    {attribute 'pytmc' := '
    pv: ACTUAL_XWIDTH;
    io: io;
    '}
    rActApertureSizeX : REAL;

    {attribute 'pytmc' := '
    pv: ACTUAL_YWIDTH;
    io: io;
    '}
    rActApertureSizeY : REAL;
    {attribute 'pytmc' := '
    pv: ACTUAL_XCENTER;
    io: io;
    '}
    rActCenterX: REAL;
    {attribute 'pytmc' := '
    pv: ACTUAL_YCENTER;
    io: io;
    '}
    rActCenterY: REAL;

    {attribute 'pytmc' := '
    pv: XCEN_SETZERO;
    io: io;
    '}
    rSetCenterX: BOOL;
    {attribute 'pytmc' := '
    pv: YCEN_SETZERO;
    io: io;
    '}
    rSetCenterY: BOOL;


    {attribute 'pytmc' := '
    pv: OPEN;
    io: io;
    field: ZNAM False
    field: ONAM True
    '}
    bOpen: BOOL;

    {attribute 'pytmc' := '
    pv: CLOSE;
    io: io;
    field: ZNAM False
    field: ONAM True
    '}
    bClose: BOOL;

    {attribute 'pytmc' := '
    pv: BLOCK;
    io: io;
    field: ZNAM False
    field: ONAM True
    '}
    bBlock: BOOL;



        //Local variables
    bInit: BOOL :=true;
    rTrig_Block: R_TRIG;
    rTrig_Open: R_TRIG;
    rTrig_Close: R_TRIG;

    //old values
    rOldReqApertureSizeX : REAL;
    rOldReqApertureSizeY : REAL;
    rOldReqCenterX: REAL;
    rOldReqCenterY: REAL;

    bExecuteMotionX: BOOL;
    bExecuteMotionY: BOOL;


    fPosBlock: LREAL;
    fPosClose: LREAL;
    fPosOpen: LREAL;

    stSetPositionOptions:ST_SetPositionOptions;
    fbSetPosition_TOP: MC_SetPosition;
    fbSetPosition_Bottom: MC_SetPosition;
    fbSetPosition_North: MC_SetPosition;
    fbSetPosition_South: MC_SetPosition;

    // For logging
    fbLogger : FB_LogMessage := (eSubsystem:=E_SubSystem.MOTION);
    tErrorPresent : R_TRIG;
    tAction : R_TRIG;
    tOverrideActivated : R_TRIG;

    FFO    :    FB_FastFault :=(
        i_DevName := 'Slits',
        i_Desc := 'Fault occurs when gaps and/or centers are not within safe margins, or PMPS mode is switched OFF',
        i_TypeCode := 16#FAA);

    AptArrayStatus AT %Q* : ST_PMPS_Aperture_IO;
    AptArrayReq AT %I* : ST_PMPS_Aperture_IO;

    bTest: BOOL;

END_VAR

ACTION ACT_BLOCK:
rTrig_Block (CLK:= bBlock);
rTrig_Open (CLK:= bOpen);
rTrig_Close (CLK:= bClose);

if (rTrig_Block.Q) THEN
    //BLOCK

    bBlock := false;
END_IF

if (rTrig_Open.Q) THEN


    bOpen := false;
END_IF

if (rTrig_Close.Q) THEN


    bClose := false;
END_IF
END_ACTION

ACTION ACT_CalculatePositions:
//check if requested center or gap has changed
//check that the requested values are within acceptable motion range
IF (rOldReqApertureSizeX <> rReqApertureSizeX) THEN
    IF (rReqApertureSizeX <= AptArrayReq.Width)  THEN
        rOldReqApertureSizeX := rReqApertureSizeX;
        bExecuteMotionX := TRUE;
        fbLogger(sMsg:='Requested new X gap.', eSevr:=TcEventSeverity.Verbose);
    ELSE
        fbLogger(sMsg:='Requested new X gap is larger than PMPS request.', eSevr:=TcEventSeverity.Verbose);
    END_IF
  //  ELSE
    //    rReqApertureSizeX := rActApertureSizeX;
END_IF

IF (rOldReqCenterX <> rReqCenterX) THEN
    rOldReqCenterX := rReqCenterX;
    bExecuteMotionX := TRUE;
    fbLogger(sMsg:='Requested new X center', eSevr:=TcEventSeverity.Verbose);
   // ELSE
      //  rReqCenterX := rActCenterX;
END_IF

IF (rOldReqApertureSizeY <> rReqApertureSizeY) THEN
    IF rReqApertureSizeY <= AptArrayReq.Height THEN
        rOldReqApertureSizeY := rReqApertureSizeY;
        bExecuteMotionY := TRUE;
        fbLogger(sMsg:='Requested new Y gap.', eSevr:=TcEventSeverity.Verbose);
    ELSE
        fbLogger(sMsg:='Requested new Y gap is larger than PMPS request.', eSevr:=TcEventSeverity.Verbose);
    END_IF
   // ELSE
       // rReqApertureSizeY := rActApertureSizeY;
END_IF

IF (rOldReqCenterY <> rReqCenterY) THEN
    rOldReqCenterY := rReqCenterY;
    bExecuteMotionY := TRUE;
    fbLogger(sMsg:='Requested new Y center.', eSevr:=TcEventSeverity.Verbose);
   // ELSE
      //  rReqCenterY := rActCenterY;
END_IF


//Calculate requested target positions from requested gap and center
fPosTopBlade := (rReqApertureSizeY/2) + (rReqCenterY + rEncoderOffsetTop) ;
fPosBottomBlade := (-1*rReqApertureSizeY/2) + (rReqCenterY+rEncoderOffsetBottom);

fPosNorthBlade := (rReqApertureSizeX/2) + (rReqCenterX + rEncoderOffsetNorth);
fPosSouthBlade := (-1*rReqApertureSizeX/2) + (rReqCenterX + rEncoderOffsetSouth);


//Calculate actual gap and center from actual stages positions
rActApertureSizeX := LREAL_TO_REAL((stNorthBlade.stAxisStatus.fActPosition - rEncoderOffsetNorth) - (stSouthBlade.stAxisStatus.fActPosition- rEncoderOffsetSouth));

rActApertureSizeY := LREAL_TO_REAL((stTopBlade.stAxisStatus.fActPosition - rEncoderOffsetTop) - (stBottomBlade.stAxisStatus.fActPosition - rEncoderOffsetBottom));

rActCenterX := LREAL_TO_REAL((((stNorthBlade.stAxisStatus.fActPosition - rEncoderOffsetNorth)  + (stSouthBlade.stAxisStatus.fActPosition - rEncoderOffsetSouth ))/2));

rActCenterY := LREAL_TO_REAL((((stTopBlade.stAxisStatus.fActPosition - rEncoderOffsetTop) + (stBottomBlade.stAxisStatus.fActPosition - rEncoderOffsetBottom))/2));



//Update PMPS Arbiter with the Actual Size and Center of the Aperture
END_ACTION

ACTION ACT_Home:

END_ACTION

ACTION ACT_Init:

//  init the motion stages parameters
IF ( bInit) THEN
    stTopBlade.bHardwareEnable := TRUE;
    stBottomBlade.bHardwareEnable := TRUE;
    stNorthBlade.bHardwareEnable := TRUE;
    stSouthBlade.bHardwareEnable := TRUE;
    stTopBlade.bPowerSelf :=TRUE;
    stBottomBlade.bPowerSelf :=TRUE;
    stNorthBlade.bPowerSelf :=TRUE;
    stSouthBlade.bPowerSelf :=TRUE;
    stTopBlade.nBrakeMode := ENUM_StageBrakeMode.NO_BRAKE;
    stBottomBlade.nBrakeMode := ENUM_StageBrakeMode.NO_BRAKE;
    stNorthBlade.nBrakeMode := ENUM_StageBrakeMode.NO_BRAKE;
    stSouthBlade.nBrakeMode := ENUM_StageBrakeMode.NO_BRAKE;
    FFO.i_DevName := i_DevName;
END_IF
END_ACTION

ACTION ACT_Motion:
// Instantiate Function block for all the blades
fbTopBlade(stMotionStage:=stTopBlade);
fbBottomBlade(stMotionStage:=stBottomBlade);
fbNorthBlade(stMotionStage:=stNorthBlade);
fbSouthBlade(stMotionStage:=stSouthBlade);

// PTP Motion for each blade
stTop.sName := 'Top';
stTop.fPosition := fPosTopBlade;
stTop.fDelta := fSmallDelta;
stTop.fVelocity := fMaxVelocity;
stTop.fAccel := fHighAccel;
stTop.fDecel := fHighAccel;

stBOTTOM.sName := 'Bottom';
stBOTTOM.fPosition := fPosBottomBlade;
stBOTTOM.fDelta := fSmallDelta;
stBOTTOM.fVelocity := fMaxVelocity;
stBOTTOM.fAccel := fHighAccel;
stBOTTOM.fDecel := fHighAccel;

stNorth.sName := 'North';
stNorth.fPosition := fPosNorthBlade;
stNorth.fDelta := fSmallDelta;
stNorth.fVelocity := fMaxVelocity;
stNorth.fAccel := fHighAccel;
stNorth.fDecel := fHighAccel;

stSouth.sName := 'South';
stSouth.fPosition := fPosSouthBlade;
stSouth.fDelta := fSmallDelta;
stSouth.fVelocity := fMaxVelocity;
stSouth.fAccel := fHighAccel;
stSouth.fDecel := fHighAccel;

IF (bExecuteMotionY) THEN
    fbTop.bExecute := fbBottom.bExecute := bExecuteMotionY;
    bExecuteMotionY:= FALSE;
END_IF

IF (bExecuteMotionX) THEN
    fbNorth.bExecute := fbSouth.bExecute := bExecuteMotionX;
    bExecuteMotionX:= FALSE;
END_IF


fbTop(
    stPositionState:=stTop,
    bMoveOk:=bMoveOk,
    stMotionStage:=stTopBlade);

fbBottom(
    stPositionState:=stBOTTOM,
    bMoveOk:=bMoveOk,
    stMotionStage:=stBottomBlade);

fbNorth(
    stPositionState:=stNorth,
    bMoveOk:=bMoveOk,
    stMotionStage:=stNorthBlade);

fbSouth(
    stPositionState:=stSouth,
    bMoveOk:=bMoveOk,
    stMotionStage:=stSouthBlade);
END_ACTION

ACTION ACT_Zero:
//ZERO BIAS

// Set Y center to zero

// Set X center to zero
(*
if (rSetCenterY)THEN
        rSetCenterY := false;
        // Set Current Position
        fbSetPosition_TOP.Position :=  stTopBlade.stAxisStatus.fActPosition - rActCenterY ;
        fbSetPosition_TOP.Execute := TRUE;
        fbSetPosition_Bottom.Position := stBottomBlade.stAxisStatus.fActPosition - rActCenterY;
        fbSetPosition_Bottom.Execute := TRUE;
END_IF

if (rSetCenterX)THEN
        rSetCenterX := false;
        // Set Current Position
        fbSetPosition_North.Position := stNorthBlade.stAxisStatus.fActPosition - rActCenterX ;
        fbSetPosition_North.Execute := TRUE;
        fbSetPosition_South.Position := stSouthBlade.stAxisStatus.fActPosition - rActCenterX ; ;
        fbSetPosition_South.Execute := TRUE;
END_IF


//Reset
if (fbSetPosition_TOP.Done ) THEN
    fbSetPosition_TOP.Execute := FALSE;
END_IF
if (fbSetPosition_Bottom.Done ) THEN
    fbSetPosition_Bottom.Execute := FALSE;
END_IF
if (fbSetPosition_North.Done ) THEN
    fbSetPosition_North.Execute := FALSE;
END_IF
if (fbSetPosition_South.Done ) THEN
    fbSetPosition_South.Execute := FALSE;
END_IF

// Set Encoder Position
//Clear position lag error
stSetPositionOptions.ClearPositionLag := TRUE;
fbSetPosition_TOP(
    Axis:=  stTopBlade.Axis ,
    Execute:= ,
    Position:= 0 ,
    Mode:= FALSE,
    Options:= stSetPositionOptions,
    Done=> ,
    Busy=> ,
    Error=> ,
    ErrorID=> );
fbSetPosition_Bottom(
    Axis:= stBottomBlade.Axis ,
    Execute:= ,
    Position:= 0 ,
    Mode:= FALSE,
    Options:= stSetPositionOptions,
    Done=> ,
    Busy=> ,
    Error=> ,
    ErrorID=> );
fbSetPosition_North(
    Axis:= stNorthBlade.Axis ,
    Execute:= ,
    Position:= 0 ,
    Mode:= FALSE,
    Options:= stSetPositionOptions,
    Done=> ,
    Busy=> ,
    Error=> ,
    ErrorID=> );
fbSetPosition_South(
    Axis:= stSouthBlade.Axis ,
    Execute:= ,
    Position:= 0 ,
    Mode:= FALSE,
    Options:= stSetPositionOptions,
    Done=> ,
    Busy=> ,
    Error=> ,
    ErrorID=> );

    *)
END_ACTION

END_FUNCTION_BLOCK

// ---- POUs/PRG_SL2K0_POWER.TcPOU
PROGRAM PRG_SL2K0_POWER
VAR
    {attribute 'pytmc' := '
        pv: SL2K0:POWER
        io: io
    '}
    {attribute 'TcLinkTo' := '.RTD_South_1.iRaw := TIIB[SL2K0-EL3202-E8]^RTD Inputs Channel 1^Value;
                              .RTD_South_1.bError := TIIB[SL2K0-EL3202-E8]^RTD Inputs Channel 1^Status^Error;
                              .RTD_South_1.bUnderrange := TIIB[SL2K0-EL3202-E8]^RTD Inputs Channel 1^Status^Underrange;
                              .RTD_South_1.bOverrange := TIIB[SL2K0-EL3202-E8]^RTD Inputs Channel 1^Status^Overrange;
                              .RTD_South_2.iRaw := TIIB[SL2K0-EL3202-E8]^RTD Inputs Channel 2^Value;
                              .RTD_South_2.bError := TIIB[SL2K0-EL3202-E8]^RTD Inputs Channel 2^Status^Error;
                              .RTD_South_2.bUnderrange := TIIB[SL2K0-EL3202-E8]^RTD Inputs Channel 2^Status^Underrange;
                              .RTD_South_2.bOverrange := TIIB[SL2K0-EL3202-E8]^RTD Inputs Channel 2^Status^Overrange;
                              .RTD_TOP_1.iRaw := TIIB[SL2K0-EL3202-E9]^RTD Inputs Channel 1^Value;
                              .RTD_TOP_1.bError := TIIB[SL2K0-EL3202-E9]^RTD Inputs Channel 1^Status^Error;
                              .RTD_TOP_1.bUnderrange := TIIB[SL2K0-EL3202-E9]^RTD Inputs Channel 1^Status^Underrange;
                              .RTD_TOP_1.bOverrange := TIIB[SL2K0-EL3202-E9]^RTD Inputs Channel 1^Status^Overrange;
                              .RTD_TOP_2.iRaw := TIIB[SL2K0-EL3202-E9]^RTD Inputs Channel 2^Value;
                              .RTD_TOP_2.bError := TIIB[SL2K0-EL3202-E9]^RTD Inputs Channel 2^Status^Error;
                              .RTD_TOP_2.bUnderrange := TIIB[SL2K0-EL3202-E9]^RTD Inputs Channel 2^Status^Underrange;
                              .RTD_TOP_2.bOverrange := TIIB[SL2K0-EL3202-E9]^RTD Inputs Channel 2^Status^Overrange;
                              .RTD_North_1.iRaw := TIIB[SL2K0-EL3202-E10]^RTD Inputs Channel 1^Value;
                              .RTD_North_1.bError := TIIB[SL2K0-EL3202-E10]^RTD Inputs Channel 1^Status^Error;
                              .RTD_North_1.bUnderrange := TIIB[SL2K0-EL3202-E10]^RTD Inputs Channel 1^Status^Underrange;
                              .RTD_North_1.bOverrange := TIIB[SL2K0-EL3202-E10]^RTD Inputs Channel 1^Status^Overrange;
                              .RTD_North_2.iRaw := TIIB[SL2K0-EL3202-E10]^RTD Inputs Channel 2^Value;
                              .RTD_North_2.bError := TIIB[SL2K0-EL3202-E10]^RTD Inputs Channel 2^Status^Error;
                              .RTD_North_2.bUnderrange := TIIB[SL2K0-EL3202-E10]^RTD Inputs Channel 2^Status^Underrange;
                              .RTD_North_2.bOverrange := TIIB[SL2K0-EL3202-E10]^RTD Inputs Channel 2^Status^Overrange;
                              .RTD_Bottom_1.iRaw := TIIB[SL2K0-EL3202-E10]^RTD Inputs Channel 1^Value;
                              .RTD_Bottom_1.bError := TIIB[SL2K0-EL3202-E10]^RTD Inputs Channel 1^Status^Error;
                              .RTD_Bottom_1.bUnderrange := TIIB[SL2K0-EL3202-E11]^RTD Inputs Channel 1^Status^Underrange;
                              .RTD_Bottom_1.bOverrange := TIIB[SL2K0-EL3202-E11]^RTD Inputs Channel 1^Status^Overrange;
                              .RTD_Bottom_2.iRaw := TIIB[SL2K0-EL3202-E11]^RTD Inputs Channel 2^Value;
                              .RTD_Bottom_2.bError := TIIB[SL2K0-EL3202-E11]^RTD Inputs Channel 2^Status^Error;
                              .RTD_Bottom_2.bUnderrange := TIIB[SL2K0-EL3202-E11]^RTD Inputs Channel 2^Status^Underrange;
                              .RTD_Bottom_2.bOverrange := TIIB[SL2K0-EL3202-E11]^RTD Inputs Channel 2^Status^Overrange;
                              .AptArrayStatus := TIIB[PMPS_PRE]^IO Outputs^AptArrayStatus^AptArrayStatus[2];
                              .AptArrayReq := TIIB[PMPS_PRE]^IO Inputs^AptArrayReq^AptArrayReq[2];
                              .fbFlowSwitch.bFlowOk := TIIB[SL2K0-EL1004-E12]^Channel 1^Input'}
    fbSL2K0: FB_SLITS_POWER;
//GET PMP Move Ok bit
// Default True until it is properly linked to PMPS bit
    bMoveOk:BOOL :=TRUE;
    {attribute 'pytmc' := '
    pv: SL2K0:POWER:GO;
    io: io;
    field: ZNAM False;
    field: ONAM True;
    '}
    bExecuteMotion:BOOL ;
    //for testing purposes only. comment-out/delete once done.
    mcPower : ARRAY [1..4] OF MC_POWER;
        (*Offsets*)
    (* Absolute encoder value at the HLS + Absolure eoncoder value at the centered beam *)
    rEncoderOffsetTop: REAL := 14.65; //15.1;
    rEncoderOffsetBottom: REAL := -12.55; //-12.2;
    rEncoderOffsetNorth: REAL :=  16.3; //15.4;
    rEncoderOffsetSouth: REAL := -12.94; //-13.4;
END_VAR


fbSL2K0.bMoveOk := bMoveOk;

fbSL2K0.rEncoderOffsetTop := rEncoderOffsetTop;
fbSL2K0.rEncoderOffsetBottom := rEncoderOffsetBottom;
fbSL2K0.rEncoderOffsetNorth := rEncoderOffsetNorth;
fbSL2K0.rEncoderOffsetSouth := rEncoderOffsetSouth;

fbSL2K0(stTopBlade:=  Main.M23,
        stBottomBlade:= Main.M25,
        stNorthBlade:=  Main.M24,
        stSouthBlade:=  Main.M22,
        bExecuteMotion:=bExecuteMotion,
        io_fbFFHWO := GVL.fbFastFaultOutput1,
        fbArbiter := GVL.fbArbiter);

fbSL2K0.M_UpdatePMPS(2);


//for testing purposes only. comment-out/delete once done.
(*mcPower[1](axis:=Main.M22.Axis, Enable:=TRUE, enable_positive:=Main.M22.bLimitForwardEnable, enable_negative:=Main.M22.bLimitBackwardEnable);
mcPower[2](axis:=Main.M23.Axis, Enable:=TRUE, enable_positive:=Main.M23.bLimitForwardEnable, enable_negative:=Main.M23.bLimitBackwardEnable);
mcPower[3](axis:=Main.M24.Axis, Enable:=TRUE, enable_positive:=Main.M24.bLimitForwardEnable, enable_negative:=Main.M24.bLimitBackwardEnable);
mcPower[4](axis:=Main.M25.Axis, Enable:=TRUE, enable_positive:=Main.M25.bLimitForwardEnable, enable_negative:=Main.M25.bLimitBackwardEnable);*)

END_PROGRAM

// ---- POUs/PRG_AT1K4_SOLID.TcPOU
PROGRAM PRG_AT1K4_SOLID
VAR
    (* TODO: use FALSE for simulation and production *)
    (* TODO: use TRUE when relying on visualization + actual hardware *)
    bDebug : BOOL := FALSE;

    nEnableMode : ENUM_StageEnableMode;

    {attribute 'pytmc' := 'pv: AT1K4:L2SI:MMS:01'}
    {attribute 'TcLinkTo' := '

        .fbRTD_1.iRaw := TIIB[AT1K4-EL3202-04]^RTD Inputs Channel 1^Value;
        .fbRTD_1.bError := TIIB[AT1K4-EL3202-04]^RTD Inputs Channel 1^Status^Error;
        .fbRTD_1.bUnderrange := TIIB[AT1K4-EL3202-04]^RTD Inputs Channel 1^Status^Underrange;
        .fbRTD_1.bOverrange := TIIB[AT1K4-EL3202-04]^RTD Inputs Channel 1^Status^Overrange;

        .fbRTD_2.iRaw := TIIB[AT1K4-EL3202-04]^RTD Inputs Channel 2^Value;
        .fbRTD_2.bError := TIIB[AT1K4-EL3202-04]^RTD Inputs Channel 2^Status^Error;
        .fbRTD_2.bUnderrange := TIIB[AT1K4-EL3202-04]^RTD Inputs Channel 2^Status^Underrange;
        .fbRTD_2.bOverrange := TIIB[AT1K4-EL3202-04]^RTD Inputs Channel 2^Status^Overrange

    '}
    fbStage1: FB_SXR_SATT_Stage;

    {attribute 'pytmc' := 'pv: AT1K4:L2SI:MMS:02'}
    {attribute 'TcLinkTo' := '

        .fbRTD_1.iRaw := TIIB[AT1K4-EL3202-03]^RTD Inputs Channel 1^Value;
        .fbRTD_1.bError := TIIB[AT1K4-EL3202-03]^RTD Inputs Channel 1^Status^Error;
        .fbRTD_1.bUnderrange := TIIB[AT1K4-EL3202-03]^RTD Inputs Channel 1^Status^Underrange;
        .fbRTD_1.bOverrange := TIIB[AT1K4-EL3202-03]^RTD Inputs Channel 1^Status^Overrange;

        .fbRTD_2.iRaw := TIIB[AT1K4-EL3202-03]^RTD Inputs Channel 2^Value;
        .fbRTD_2.bError := TIIB[AT1K4-EL3202-03]^RTD Inputs Channel 2^Status^Error;
        .fbRTD_2.bUnderrange := TIIB[AT1K4-EL3202-03]^RTD Inputs Channel 2^Status^Underrange;
        .fbRTD_2.bOverrange := TIIB[AT1K4-EL3202-03]^RTD Inputs Channel 2^Status^Overrange

    '}
    fbStage2: FB_SXR_SATT_Stage;

    {attribute 'pytmc' := 'pv: AT1K4:L2SI:MMS:03'}
    {attribute 'TcLinkTo' := '

        .fbRTD_1.iRaw := TIIB[AT1K4-EL3202-02]^RTD Inputs Channel 1^Value;
        .fbRTD_1.bError := TIIB[AT1K4-EL3202-02]^RTD Inputs Channel 1^Status^Error;
        .fbRTD_1.bUnderrange := TIIB[AT1K4-EL3202-02]^RTD Inputs Channel 1^Status^Underrange;
        .fbRTD_1.bOverrange := TIIB[AT1K4-EL3202-02]^RTD Inputs Channel 1^Status^Overrange;

        .fbRTD_2.iRaw := TIIB[AT1K4-EL3202-02]^RTD Inputs Channel 2^Value;
        .fbRTD_2.bError := TIIB[AT1K4-EL3202-02]^RTD Inputs Channel 2^Status^Error;
        .fbRTD_2.bUnderrange := TIIB[AT1K4-EL3202-02]^RTD Inputs Channel 2^Status^Underrange;
        .fbRTD_2.bOverrange := TIIB[AT1K4-EL3202-02]^RTD Inputs Channel 2^Status^Overrange
    '}
    fbStage3: FB_SXR_SATT_Stage;

    {attribute 'pytmc' := 'pv: AT1K4:L2SI:MMS:04'}
    {attribute 'TcLinkTo' := '

        .fbRTD_1.iRaw := TIIB[AT1K4-EL3202-01]^RTD Inputs Channel 1^Value;
        .fbRTD_1.bError := TIIB[AT1K4-EL3202-01]^RTD Inputs Channel 1^Status^Error;
        .fbRTD_1.bUnderrange := TIIB[AT1K4-EL3202-01]^RTD Inputs Channel 1^Status^Underrange;
        .fbRTD_1.bOverrange := TIIB[AT1K4-EL3202-01]^RTD Inputs Channel 1^Status^Overrange;

        .fbRTD_2.iRaw := TIIB[AT1K4-EL3202-01]^RTD Inputs Channel 2^Value;
        .fbRTD_2.bError := TIIB[AT1K4-EL3202-01]^RTD Inputs Channel 2^Status^Error;
        .fbRTD_2.bUnderrange := TIIB[AT1K4-EL3202-01]^RTD Inputs Channel 2^Status^Underrange;
        .fbRTD_2.bOverrange := TIIB[AT1K4-EL3202-01]^RTD Inputs Channel 2^Status^Overrange
    '}
    fbStage4: FB_SXR_SATT_Stage;

    fbStateSetup: FB_StateSetupHelper;
    stDefaultGood: ST_PositionState := (
        fDelta := 0.2,
        fVelocity := 10,
        bMoveOk := TRUE,
        bValid := TRUE
    );
    fbBadStateSetup: FB_StateSetupHelper;
    stDefaultBad: ST_PositionState := (
        fPosition := 500,
        fDelta := 0.2,
        fVelocity := 10,
        bMoveOk := FALSE,
        bValid := FALSE

    );
END_VAR

// M26, Axis 26
// M27, Axis 27
// M28, Axis 28
// M29, Axis 29

IF bDebug THEN
    // NEVER: checkouts with the TwinCAT NC GUI.
    nEnableMode := ENUM_StageEnableMode.NEVER;
ELSE
    // ALWAYS: want active position correction at all times
    nEnableMode := ENUM_StageEnableMode.ALWAYS;
END_IF

(*
    Important note

    Traveler	EPICS	Stage		NC	Location
    Axis 4		MMS:01	fbStage1	26	Downstream
    Axis 3		MMS:02	fbStage2	27
    Axis 2		MMS:03	fbStage3	28
    Axis 1		MMS:04	fbStage4	29	Upstream
*)

fbStateSetup(stPositionState:=stDefaultGood, bSetDefault:=TRUE);
fbBadStateSetup(stPositionState:=stDefaultBad, bSetDefault:=TRUE);

(* State setup - stage 1 *)
(* Downstream-most MMS:01 - TRAVELER AXIS 4 *)
fbStateSetup(stPositionState:=fbStage1.stOut, sName:='Out', fPosition:=22.70);
fbStateSetup(stPositionState:=fbStage1.stFilter1, sName:='(1) 25 um C', fPosition:=40.5, sPmpsState:='AT1K4:L2SI-RTD');
fbStage1.arrFilters[1].fFilterThickness_um := 25;
fbStage1.arrFilters[1].sFilterMaterial     := 'C';
fbStateSetup(stPositionState:=fbStage1.stFilter2, sName:='(2) 50 um C', fPosition:=56.0);
fbStage1.arrFilters[2].fFilterThickness_um := 50;
fbStage1.arrFilters[2].sFilterMaterial     := 'C';
fbStateSetup(stPositionState:=fbStage1.stFilter3, sName:='(3) 100 um C', fPosition:=72.0);
fbStage1.arrFilters[3].fFilterThickness_um := 100;
fbStage1.arrFilters[3].sFilterMaterial     := 'C';
fbStateSetup(stPositionState:=fbStage1.stFilter4, sName:='(4) 320 um Si', fPosition:=87.5);
fbStage1.arrFilters[4].fFilterThickness_um := 320;
fbStage1.arrFilters[4].sFilterMaterial     := 'Si';
fbStateSetup(stPositionState:=fbStage1.stFilter5, sName:='(5) 160 um Si', fPosition:=102.5);
fbStage1.arrFilters[5].fFilterThickness_um := 160;
fbStage1.arrFilters[5].sFilterMaterial     := 'Si';
fbStateSetup(stPositionState:=fbStage1.stFilter6, sName:='(6) 80 um Si', fPosition:=117.5);
fbStage1.arrFilters[6].fFilterThickness_um := 80;
fbStage1.arrFilters[6].sFilterMaterial     := 'Si';
fbStateSetup(stPositionState:=fbStage1.stFilter7, sName:='(7) 40 um Si', fPosition:=135.5);
fbStage1.arrFilters[7].fFilterThickness_um := 40;
fbStage1.arrFilters[7].sFilterMaterial     := 'Si';
fbStateSetup(stPositionState:=fbStage1.stFilter8, sName:='(8) 20 um Si', fPosition:=150.5);
fbStage1.arrFilters[8].fFilterThickness_um := 20;
fbStage1.arrFilters[8].sFilterMaterial     := 'Si';

fbStage1(stAxis:=Main.M26, nEnableMode:=nEnableMode, fbFFHWO:=GVL.fbFastFaultOutput2, bEnable:=TRUE, sDeviceName:='AT1K4:L2SI');

(* State setup - stage 2 *)
(* MMS:02 - 2nd downstream-most - TRAVELER AXIS 3 *)
fbStateSetup(stPositionState:=fbStage2.stOut, sName:='Out', fPosition:=24.00);
fbBadStateSetup(stPositionState:=fbStage2.stFilter1, sName:='Filter 1', sPmpsState:='AT1K4:L2SI-RTD');
fbStage2.arrFilters[1].fFilterThickness_um := 0;
fbStage2.arrFilters[1].sFilterMaterial     := '';
fbBadStateSetup(stPositionState:=fbStage2.stFilter2, sName:='Filter 2');
fbStage2.arrFilters[2].fFilterThickness_um := 0;
fbStage2.arrFilters[2].sFilterMaterial     := '';
fbBadStateSetup(stPositionState:=fbStage2.stFilter3, sName:='Filter 3');
fbStage2.arrFilters[3].fFilterThickness_um := 0;
fbStage2.arrFilters[3].sFilterMaterial     := '';
fbBadStateSetup(stPositionState:=fbStage2.stFilter4, sName:='Filter 4');
fbStage2.arrFilters[4].fFilterThickness_um := 0;
fbStage2.arrFilters[4].sFilterMaterial     := '';
fbStateSetup(stPositionState:=fbStage2.stFilter5, sName:='(5) 50 um C', fPosition:=103.0);
fbStage2.arrFilters[5].fFilterThickness_um := 50;
fbStage2.arrFilters[5].sFilterMaterial     := 'C';
fbStateSetup(stPositionState:=fbStage2.stFilter6, sName:='(6) 25 um C', fPosition:=118.75);
fbStage2.arrFilters[6].fFilterThickness_um := 25;
fbStage2.arrFilters[6].sFilterMaterial     := 'C';
fbStateSetup(stPositionState:=fbStage2.stFilter7, sName:='(7) 12 um C', fPosition:=133.0);
fbStage2.arrFilters[7].fFilterThickness_um := 12;
fbStage2.arrFilters[7].sFilterMaterial     := 'C';
fbStateSetup(stPositionState:=fbStage2.stFilter8, sName:='(8) 10 um Si', fPosition:=147.0);
fbStage2.arrFilters[8].fFilterThickness_um := 10;
fbStage2.arrFilters[8].sFilterMaterial     := 'Si';

fbStage2(stAxis:=Main.M27, nEnableMode:=nEnableMode, fbFFHWO:=GVL.fbFastFaultOutput2, bEnable:=TRUE, sDeviceName:='AT1K4:L2SI');

(* State setup - stage 3 *)
(* MMS:03 - 2nd upstream-most - TRAVELER AXIS 2 *)
fbStateSetup(stPositionState:=fbStage3.stOut, sName:='Out', fPosition:=23.24);
fbBadStateSetup(stPositionState:=fbStage3.stFilter1, sName:='Filter 1', sPmpsState:='AT1K4:L2SI-RTD');
fbStage3.arrFilters[1].fFilterThickness_um := 0;
fbStage3.arrFilters[1].sFilterMaterial     := '';
fbBadStateSetup(stPositionState:=fbStage3.stFilter2, sName:='Filter 2');
fbStage3.arrFilters[2].fFilterThickness_um := 0;
fbStage3.arrFilters[2].sFilterMaterial     := '';
fbBadStateSetup(stPositionState:=fbStage3.stFilter3, sName:='Filter 3');
fbStage3.arrFilters[3].fFilterThickness_um := 0;
fbStage3.arrFilters[3].sFilterMaterial     := '';
fbBadStateSetup(stPositionState:=fbStage3.stFilter4, sName:='Filter 4');
fbStage3.arrFilters[4].fFilterThickness_um := 0;
fbStage3.arrFilters[4].sFilterMaterial     := '';
fbBadStateSetup(stPositionState:=fbStage3.stFilter5, sName:='Filter 5');
fbStage3.arrFilters[5].fFilterThickness_um := 0;
fbStage3.arrFilters[5].sFilterMaterial     := '';
fbStateSetup(stPositionState:=fbStage3.stFilter6, sName:='(6) 25 um C', fPosition:=119.5);
fbStage3.arrFilters[6].fFilterThickness_um := 25;
fbStage3.arrFilters[6].sFilterMaterial     := 'C';
fbStateSetup(stPositionState:=fbStage3.stFilter7, sName:='(7) 12 um C', fPosition:=135.0);
fbStage3.arrFilters[7].fFilterThickness_um := 12;
fbStage3.arrFilters[7].sFilterMaterial     := 'C';
fbStateSetup(stPositionState:=fbStage3.stFilter8, sName:='(8) 6 um C', fPosition:=147.5);
fbStage3.arrFilters[8].fFilterThickness_um := 6;
fbStage3.arrFilters[8].sFilterMaterial     := 'C';

fbStage3(stAxis:=Main.M28, nEnableMode:=nEnableMode, fbFFHWO:=GVL.fbFastFaultOutput2, bEnable:=TRUE, sDeviceName:='AT1K4:L2SI');

(* State setup - stage 4 *)
(* MMS:04 - upstream-most - TRAVELER AXIS 1 *)
fbStateSetup(stPositionState:=fbStage4.stOut, sName:='Out', fPosition:=23.44);
fbBadStateSetup(stPositionState:=fbStage4.stFilter1, sName:='Filter 1', sPmpsState:='AT1K4:L2SI-RTD');
fbStage4.arrFilters[1].fFilterThickness_um := 0;
fbStage4.arrFilters[1].sFilterMaterial     := '';
fbBadStateSetup(stPositionState:=fbStage4.stFilter2, sName:='Filter 2');
fbStage4.arrFilters[2].fFilterThickness_um := 0;
fbStage4.arrFilters[2].sFilterMaterial     := '';
fbBadStateSetup(stPositionState:=fbStage4.stFilter3, sName:='Filter 3');
fbStage4.arrFilters[3].fFilterThickness_um := 0;
fbStage4.arrFilters[3].sFilterMaterial     := '';
fbStateSetup(stPositionState:=fbStage4.stFilter4, sName:='(4) 12 um C', fPosition:=85.5);
fbStage4.arrFilters[4].fFilterThickness_um := 12;
fbStage4.arrFilters[4].sFilterMaterial     := 'C';
fbStateSetup(stPositionState:=fbStage4.stFilter5, sName:='(5) 6 um C', fPosition:=100.5);
fbStage4.arrFilters[5].fFilterThickness_um := 6;
fbStage4.arrFilters[5].sFilterMaterial     := 'C';
fbStateSetup(stPositionState:=fbStage4.stFilter6, sName:='(6) 3 um C', fPosition:=116.0);
fbStage4.arrFilters[6].fFilterThickness_um := 3;
fbStage4.arrFilters[6].sFilterMaterial     := 'C';
fbStateSetup(stPositionState:=fbStage4.stFilter7, sName:='(7) 3 um C', fPosition:=132.0);
fbStage4.arrFilters[7].fFilterThickness_um := 3;
fbStage4.arrFilters[7].sFilterMaterial     := 'C';
fbStateSetup(stPositionState:=fbStage4.stFilter8, sName:='(8) 0.2 um Al', fPosition:=147.0);
fbStage4.arrFilters[8].fFilterThickness_um := 0.2;
fbStage4.arrFilters[8].sFilterMaterial     := 'Al';

fbStage4(stAxis:=Main.M29, nEnableMode:=nEnableMode, fbFFHWO:=GVL.fbFastFaultOutput2, bEnable:=TRUE, sDeviceName:='AT1K4:L2SI');

GVL.rCurTrans[PMPS.K_Attenuators.AT1K4].nTran := LREAL_TO_REAL(
    fbStage1.fTransmission *
    fbStage2.fTransmission *
    fbStage3.fTransmission *
    fbStage4.fTransmission
);

END_PROGRAM

// ---- POUs/PRG_IM1K4_XTES.TcPOU
PROGRAM PRG_IM1K4_XTES
VAR
    {attribute 'pytmc' := 'pv: IM1K4:XTES'}
    {attribute 'TcLinkTo' := '.bZoomEndFwd := TIIB[IM1K4-EL1088-E5]^Channel 1^Input;
                              .bZoomEndBwd := TIIB[IM1K4-EL1088-E5]^Channel 2^Input;
                              .bFocusEndFwd := TIIB[IM1K4-EL1088-E5]^Channel 3^Input;
                              .bFocusEndBwd := TIIB[IM1K4-EL1088-E5]^Channel 4^Input;
                              .fbOpal.bOpalPower := TIIB[IM1K4-EL2004-E2]^Channel 2^Output;
                              .fbLED.bLedPower := TIIB[IM1K4-EL2004-E2]^Channel 3^Output;
                              .fbFlowSwitch.bFlowOk := TIIB[ST1K4-EL1004-E5]^Channel 2^Input'} // same as PC1K4
    fbIM1K4: FB_XPIM;
    fbStateSetup: FB_StateSetupHelper;
    stDefault: ST_PositionState := (
        fVelocity := 1,
        bMoveOk := TRUE,
        bValid := TRUE
    );
    {attribute 'TcLinkTo' := '.Status := TIIB[IM1K4-EL6002-E6]^COM TxPDO-Map Inputs Channel 1^Status;
                              .D[0] := TIIB[IM1K4-EL6002-E6]^COM TxPDO-Map Inputs Channel 1^Data In 0;
                              .D[1] := TIIB[IM1K4-EL6002-E6]^COM TxPDO-Map Inputs Channel 1^Data In 1;
                              .D[2] := TIIB[IM1K4-EL6002-E6]^COM TxPDO-Map Inputs Channel 1^Data In 2;
                              .D[3] := TIIB[IM1K4-EL6002-E6]^COM TxPDO-Map Inputs Channel 1^Data In 3;
                              .D[4] := TIIB[IM1K4-EL6002-E6]^COM TxPDO-Map Inputs Channel 1^Data In 4;
                              .D[5] := TIIB[IM1K4-EL6002-E6]^COM TxPDO-Map Inputs Channel 1^Data In 5;
                              .D[6] := TIIB[IM1K4-EL6002-E6]^COM TxPDO-Map Inputs Channel 1^Data In 6;
                              .D[7] := TIIB[IM1K4-EL6002-E6]^COM TxPDO-Map Inputs Channel 1^Data In 7;
                              .D[8] := TIIB[IM1K4-EL6002-E6]^COM TxPDO-Map Inputs Channel 1^Data In 8;
                              .D[9] := TIIB[IM1K4-EL6002-E6]^COM TxPDO-Map Inputs Channel 1^Data In 9;
                              .D[10] := TIIB[IM1K4-EL6002-E6]^COM TxPDO-Map Inputs Channel 1^Data In 10;
                              .D[11] := TIIB[IM1K4-EL6002-E6]^COM TxPDO-Map Inputs Channel 1^Data In 11;
                              .D[12] := TIIB[IM1K4-EL6002-E6]^COM TxPDO-Map Inputs Channel 1^Data In 12;
                              .D[13] := TIIB[IM1K4-EL6002-E6]^COM TxPDO-Map Inputs Channel 1^Data In 13;
                              .D[14] := TIIB[IM1K4-EL6002-E6]^COM TxPDO-Map Inputs Channel 1^Data In 14;
                              .D[15] := TIIB[IM1K4-EL6002-E6]^COM TxPDO-Map Inputs Channel 1^Data In 15;
                              .D[16] := TIIB[IM1K4-EL6002-E6]^COM TxPDO-Map Inputs Channel 1^Data In 16;
                              .D[17] := TIIB[IM1K4-EL6002-E6]^COM TxPDO-Map Inputs Channel 1^Data In 17;
                              .D[18] := TIIB[IM1K4-EL6002-E6]^COM TxPDO-Map Inputs Channel 1^Data In 18;
                              .D[19] := TIIB[IM1K4-EL6002-E6]^COM TxPDO-Map Inputs Channel 1^Data In 19;
                              .D[20] := TIIB[IM1K4-EL6002-E6]^COM TxPDO-Map Inputs Channel 1^Data In 20;
                              .D[21] := TIIB[IM1K4-EL6002-E6]^COM TxPDO-Map Inputs Channel 1^Data In 21'}
    stEL6In AT %I*: EL6InData22b;
    {attribute 'TcLinkTo' := '.Ctrl := TIIB[IM1K4-EL6002-E6]^COM RxPDO-Map Outputs Channel 1^Ctrl;
                              .D[0] := TIIB[IM1K4-EL6002-E6]^COM RxPDO-Map Outputs Channel 1^Data Out 0;
                              .D[1] := TIIB[IM1K4-EL6002-E6]^COM RxPDO-Map Outputs Channel 1^Data Out 1;
                              .D[2] := TIIB[IM1K4-EL6002-E6]^COM RxPDO-Map Outputs Channel 1^Data Out 2;
                              .D[3] := TIIB[IM1K4-EL6002-E6]^COM RxPDO-Map Outputs Channel 1^Data Out 3;
                              .D[4] := TIIB[IM1K4-EL6002-E6]^COM RxPDO-Map Outputs Channel 1^Data Out 4;
                              .D[5] := TIIB[IM1K4-EL6002-E6]^COM RxPDO-Map Outputs Channel 1^Data Out 5;
                              .D[6] := TIIB[IM1K4-EL6002-E6]^COM RxPDO-Map Outputs Channel 1^Data Out 6;
                              .D[7] := TIIB[IM1K4-EL6002-E6]^COM RxPDO-Map Outputs Channel 1^Data Out 7;
                              .D[8] := TIIB[IM1K4-EL6002-E6]^COM RxPDO-Map Outputs Channel 1^Data Out 8;
                              .D[9] := TIIB[IM1K4-EL6002-E6]^COM RxPDO-Map Outputs Channel 1^Data Out 9;
                              .D[10] := TIIB[IM1K4-EL6002-E6]^COM RxPDO-Map Outputs Channel 1^Data Out 10;
                              .D[11] := TIIB[IM1K4-EL6002-E6]^COM RxPDO-Map Outputs Channel 1^Data Out 11;
                              .D[12] := TIIB[IM1K4-EL6002-E6]^COM RxPDO-Map Outputs Channel 1^Data Out 12;
                              .D[13] := TIIB[IM1K4-EL6002-E6]^COM RxPDO-Map Outputs Channel 1^Data Out 13;
                              .D[14] := TIIB[IM1K4-EL6002-E6]^COM RxPDO-Map Outputs Channel 1^Data Out 14;
                              .D[15] := TIIB[IM1K4-EL6002-E6]^COM RxPDO-Map Outputs Channel 1^Data Out 15;
                              .D[16] := TIIB[IM1K4-EL6002-E6]^COM RxPDO-Map Outputs Channel 1^Data Out 16;
                              .D[17] := TIIB[IM1K4-EL6002-E6]^COM RxPDO-Map Outputs Channel 1^Data Out 17;
                              .D[18] := TIIB[IM1K4-EL6002-E6]^COM RxPDO-Map Outputs Channel 1^Data Out 18;
                              .D[19] := TIIB[IM1K4-EL6002-E6]^COM RxPDO-Map Outputs Channel 1^Data Out 19;
                              .D[20] := TIIB[IM1K4-EL6002-E6]^COM RxPDO-Map Outputs Channel 1^Data Out 20;
                              .D[21] := TIIB[IM1K4-EL6002-E6]^COM RxPDO-Map Outputs Channel 1^Data Out 21'}
    stEL6Out AT %Q*: EL6OutData22b;

    {attribute 'pytmc' := '
        pv: IM1K4:SCRP:LED:01:PWR
        io: io
        field: ZNAM OFF
        field: ONAM ON
    '}
    {attribute 'TcLinkTo' := 'TIIB[IM1K4-EL2004-E2]^Channel 4^Output'}
    bIM1K4_SCRP_LED_01 AT %Q*: BOOL;
END_VAR


fbStateSetup(stPositionState:=stDefault, bSetDefault:=TRUE);

fbStateSetup(stPositionState:=fbIM1K4.stOut, fPosition:=0, sPmpsState:='IM1K4:XTES-OUT');
fbStateSetup(stPositionState:=fbIM1K4.stYag, fPosition:=-88.87, sPmpsState:='IM1K4:XTES-YAG');
fbStateSetup(stPositionState:=fbIM1K4.stDiamond, fPosition:=-58.87, sPmpsState:='IM1K4:XTES-DIAMOND');
fbStateSetup(stPositionState:=fbIM1K4.stReticle, fPosition:=-28.87, sPmpsState:='IM1K4:XTES-RETICLE');

fbIM1K4(
    fbFFHWO := GVL.fbFastFaultOutput2,
    fbArbiter := GVL.fbArbiter2,
    stYStage := Main.M30,
    stZoomStage := Main.M31,
    stFocusStage := Main.M32,
    stEl6In := stEL6In,
    stEl6Out := stEl6Out,
    sDeviceName := 'IM1K4:XTES',
    sTransitionKey := 'IM1K4:XTES-TRANSITION',
    bEnableMotion := TRUE,
    bEnableBeamParams := TRUE,
    bEnablePositionLimits := TRUE,
);

END_PROGRAM

// ---- POUs/PRG_ST1K4_TEST.TcPOU
PROGRAM PRG_ST1K4_TEST
VAR
    fbMotion: FB_MotionStage;

    {attribute 'pytmc' := '
        pv: ST1K4:TEST:MMS
        astPositionState.array: 1..2
    '}
    fbStates: FB_PositionState1D;

    fbStateSetup: FB_StateSetupHelper;
    stDefault: ST_PositionState := (
        fDelta := 1,
        fVelocity := 5,
        bMoveOk := TRUE,
        bValid := TRUE
    );
    astPositionState: ARRAY[1..GeneralConstants.MAX_STATES] OF ST_PositionState;

    {attribute 'pytmc' := '
        pv: ST1K4:TEST:MMS:STATE:GET
        io: i
    '}
    eEnumGet: E_EpicsInOut;
    {attribute 'pytmc' := '
        pv: ST1K4:TEST:MMS:STATE:SET
        io: io
    '}
    eEnumSet: E_EpicsInOut;

    bST3K4_in: BOOL;

    {attribute 'pytmc' := '
        pv: ST1K4:TEST:MMS:STATE:ST3K4_AUTO
        io: io
    '}
    bST3K4_auto: BOOL := TRUE;

    {attribute 'pytmc' := '
        pv: ST1K4:TEST:FSW
    '}
    {attribute 'TcLinkTo' := '.bFlowOk := TIIB[ST1K4-EL1004-E5]^Channel 1^Input'}
    fbFlowSwitch: FB_XTES_Flowswitch;


    // Raw encoder PMPS VETO
      {attribute 'TcLinkTo' := 'TIIB[ST1K4-EL5042-E6]^FB Inputs Channel 1^Position'}
    nRawEncoderULINT AT %I*: ULINT;
END_VAR


// M33, Axis 33
Main.M33.nEnableMode := ENUM_StageEnableMode.DURING_MOTION;
Main.M33.bHardwareEnable:= TRUE;
Main.M33.bPowerSelf := TRUE;
Main.M33.nBrakeMode := ENUM_StageBrakeMode.IF_ENABLED;
fbMotion(stMotionStage:=Main.M33);

// States
fbStateSetup(stPositionState:=stDefault, bSetDefault:=TRUE);

fbStateSetup(stPositionState:=astPositionState[E_EpicsInOut.IN], sName:='IN', fPosition:=2);
fbStateSetup(stPositionState:=astPositionState[E_EpicsInOut.OUT], sName:='OUT', fPosition:=40.9);

fbStates(
    stMotionStage:=Main.M33,
    astPositionState:=astPositionState,
    eEnumSet:=eEnumSet,
    eEnumGet:=eEnumGet,
    bEnable:=TRUE,
);

bST3K4_in := PMPS_GVL.stCurrentBeamParameters.aVetoDevices[PMPS.K_Stopper.ST3K4];


IF bST3K4_auto THEN
    IF bST3K4_in AND eEnumGet <> E_EpicsInOut.IN THEN
        eEnumSet := ENUM_EpicsInOut.IN;
{*    ELSIF NOT bST3K4_in AND eEnumGet <> E_EpicsInOut.OUT THEN
        eEnumSet := ENUM_EpicsInOut.OUT;
 *}   END_IF
END_IF

fbFlowSwitch();

// For PMPS Veto
    GVL.PMPS_ST1K4_Y_ENC := TO_UDINT(nRawEncoderULINT);

END_PROGRAM

// ---- POUs/PRG_OTHER.TcPOU
PROGRAM PRG_OTHER
// A Program for implementing devices with minimal interaction.
VAR
    {attribute 'pytmc' := 'pv: PC1K0:XTES:FSW'}
    {attribute 'TcLinkTo' := '.bFlowOk := TIIB[IM1K0-EL1004]^Channel 1^Input'}
    fbPC1K0FlowSwitch : FB_XTES_Flowswitch;

    {attribute 'pytmc' := 'pv: PC1K4:XTES:FSW'}
    {attribute 'TcLinkTo' := '.bFlowOk := TIIB[ST1K4-EL1004-E5]^Channel 2^Input'}
    fbPC1K4FlowSwitch : FB_XTES_Flowswitch;
END_VAR

fbPC1K0FlowSwitch();
fbPC1K4FlowSwitch();

END_PROGRAM

// ---- POUs/PRG_3_PMPS_POST.TcPOU
PROGRAM PRG_3_PMPS_POST
VAR
    fbArbiterIO: FB_SubSysToArbiter_IO;
    fb_vetoArbiter_K4: FB_VetoArbiter;
    fb_vetoArbiter_K3: FB_VetoArbiter;
    ff3_ff2_link: FB_FastFault := (i_xAutoReset := TRUE, i_DevName := 'FF3 to FF2 Link', i_Desc := 'This is virtual FF3 fault, Please check the Group 3 faulting device ', i_TypeCode := 16#9999);

    bM1K1_Veto_IN: BOOL;
    bM1K3_Veto_IN: BOOL;
    bM1K3_Veto_OUT: BOOL;
END_VAR

// create MR1K1 as veto for K4 lines
bM1K1_Veto_IN := NOT PMPS_GVL.stCurrentBeamParameters.aVetoDevices[PMPS.K_Stopper.MR1K1_OUT]
                AND PMPS_GVL.stCurrentBeamParameters.aVetoDevices[PMPS.K_Stopper.MR1K1_IN];
// create MR1K3 as veto for K4 lines
bM1K3_Veto_IN := NOT PMPS_GVL.stCurrentBeamParameters.aVetoDevices[PMPS.K_Stopper.MR1K3_OUT]
                AND PMPS_GVL.stCurrentBeamParameters.aVetoDevices[PMPS.K_Stopper.MR1K3_IN];
// create MR1K3 as veto for IM1K3
bM1K3_Veto_OUT := NOT PMPS_GVL.stCurrentBeamParameters.aVetoDevices[PMPS.K_Stopper.MR1K3_IN]
                 AND PMPS_GVL.stCurrentBeamParameters.aVetoDevices[PMPS.K_Stopper.MR1K3_OUT];




//create a preemptive request from Arbiter 2 in Arbiter 1
fb_vetoArbiter_K4(bVeto:=bM1K1_Veto_IN OR bM1K3_Veto_IN,
                HigherAuthority := GVL.fbArbiter,
                LowerAuthority := GVL.fbArbiter2,
                FFO := GVL.fbFastFaultOutput2);
fb_vetoArbiter_K3(bVeto:=(bM1K1_Veto_IN OR bM1K3_VETO_OUT),
                HigherAuthority := GVL.fbArbiter,
                LowerAuthority := GVL.fbArbiter3,
                FFO := GVL.fbFastFaultOutput3);


GVL.fbFastFaultOutput1.Execute();

GVL.fbFastFaultOutput2.Execute(i_xVeto:=bM1K1_Veto_IN OR bM1K3_Veto_IN);

GVL.fbFastFaultOutput3.Execute(i_xVeto:=(bM1K1_Veto_IN OR bM1K3_Veto_OUT));

fbArbiterIO(
    Arbiter:=GVL.fbArbiter,
    fbFFHWO:=GVL.fbFastFaultOutput1);

ff3_ff2_link(
    io_fbFFHWO := GVL.fbFastFaultOutput2,
    i_xOK := GVL.fbFastFaultOutput3.q_xFastFaultOut);

END_PROGRAM

// ---- POUs/PRG_4_LOG.TcPOU
PROGRAM PRG_4_LOG
VAR
    fbLogHandler: FB_LogHandler;
END_VAR

fbLogHandler();

END_PROGRAM
